TYPE ST_MotorValues :
STRUCT
	iEncoderPosition 	: INT;
	rSpeed				: REAL;
	bOverheat			: BOOL;
END_STRUCT
END_TYPE

(* stored: Version 1.1.0.1, ProductVersion 3.1.4024.9
   DUT ST_MotorValues: Id {d43f7281-4e0d-4fd3-b2eb-381d860f5bff} *)
